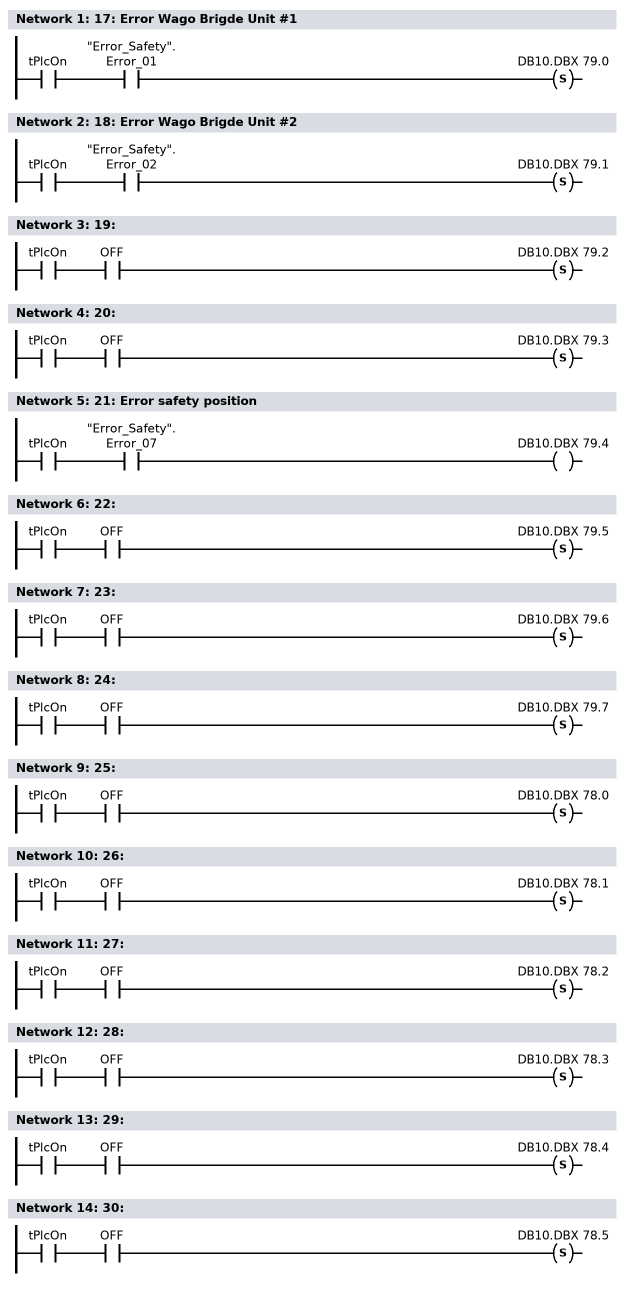
[picture p24: Errors_017-032_GEN2 networks 1-14]
NETWORK
TITLE = 17: Error Wago Brigde Unit #1
      A     "tPlcOn";
      A     "Error_Safety".Error_01;
      S     DB10.DBX 79.0;
NETWORK
TITLE = 18: Error Wago Brigde Unit #2
      A     "tPlcOn";
      A     "Error_Safety".Error_02;
      S     DB10.DBX 79.1;
NETWORK
TITLE = 19:
      A     "tPlcOn";
      A     "OFF";
      S     DB10.DBX 79.2;
NETWORK
TITLE = 20:
      A     "tPlcOn";
      A     "OFF";
      S     DB10.DBX 79.3;
NETWORK
TITLE = 21: Error safety position
      A     "tPlcOn";
      A     "Error_Safety".Error_07;
      =     DB10.DBX 79.4;
NETWORK
TITLE = 22:
      A     "tPlcOn";
      A     "OFF";
      S     DB10.DBX 79.5;
NETWORK
TITLE = 23:
      A     "tPlcOn";
      A     "OFF";
      S     DB10.DBX 79.6;
NETWORK
TITLE = 24:
      A     "tPlcOn";
      A     "OFF";
      S     DB10.DBX 79.7;
NETWORK
TITLE = 25:
      A     "tPlcOn";
      A     "OFF";
      S     DB10.DBX 78.0;
NETWORK
TITLE = 26:
      A     "tPlcOn";
      A     "OFF";
      S     DB10.DBX 78.1;
NETWORK
TITLE = 27:
      A     "tPlcOn";
      A     "OFF";
      S     DB10.DBX 78.2;
NETWORK
TITLE = 28:
      A     "tPlcOn";
      A     "OFF";
      S     DB10.DBX 78.3;
NETWORK
TITLE = 29:
      A     "tPlcOn";
      A     "OFF";
      S     DB10.DBX 78.4;
NETWORK
TITLE = 30:
      A     "tPlcOn";
      A     "OFF";
      S     DB10.DBX 78.5;
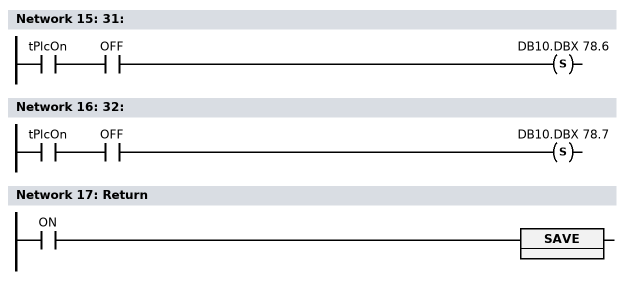
NETWORK
TITLE = 31:
      A     "tPlcOn";
      A     "OFF";
      S     DB10.DBX 78.6;
NETWORK
TITLE = 32:
      A     "tPlcOn";
      A     "OFF";
      S     DB10.DBX 78.7;
NETWORK
TITLE = Return
      A     "ON";
      SAVE;
END_FUNCTION

FUNCTION "Errors_033-048_NET" : VOID	// FC 44
TITLE = Errors NET
VERSION : 0.1
BEGIN
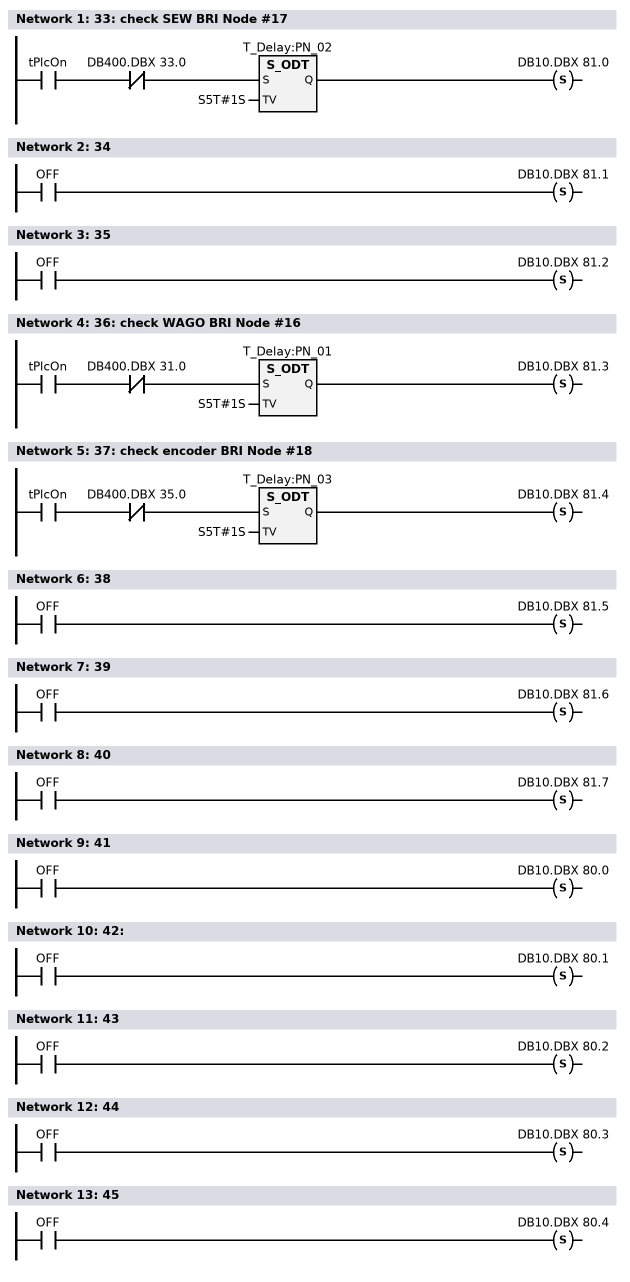
NETWORK
TITLE = 33: check SEW BRI Node #17
      A     "tPlcOn";
      AN    DB400.DBX 33.0;
      L     S5T#1S;
      SD    "T_Delay:PN_02";
      NOP   0;
      NOP   0;
      NOP   0;
      A     "T_Delay:PN_02";
      S     DB10.DBX 81.0;
NETWORK
TITLE = 34
      A     "OFF";
      S     DB10.DBX 81.1;
NETWORK
TITLE = 35
      A     "OFF";
      S     DB10.DBX 81.2;
NETWORK
TITLE = 36: check WAGO BRI Node #16
      A     "tPlcOn";
      AN    DB400.DBX 31.0;
      L     S5T#1S;
      SD    "T_Delay:PN_01";
      NOP   0;
      NOP   0;
      NOP   0;
      A     "T_Delay:PN_01";
      S     DB10.DBX 81.3;
NETWORK
TITLE = 37: check encoder BRI Node #18
      A     "tPlcOn";
      AN    DB400.DBX 35.0;
      L     S5T#1S;
      SD    "T_Delay:PN_03";
      NOP   0;
      NOP   0;
      NOP   0;
      A     "T_Delay:PN_03";
      S     DB10.DBX 81.4;
NETWORK
TITLE = 38
      A     "OFF";
      S     DB10.DBX 81.5;
NETWORK
TITLE = 39
      A     "OFF";
      S     DB10.DBX 81.6;
NETWORK
TITLE = 40
      A     "OFF";
      S     DB10.DBX 81.7;
NETWORK
TITLE = 41
      A     "OFF";
      S     DB10.DBX 80.0;
NETWORK
TITLE = 42:
      A     "OFF";
      S     DB10.DBX 80.1;
NETWORK
TITLE = 43
      A     "OFF";
      S     DB10.DBX 80.2;
NETWORK
TITLE = 44
      A     "OFF";
      S     DB10.DBX 80.3;
NETWORK
TITLE = 45
      A     "OFF";
      S     DB10.DBX 80.4;
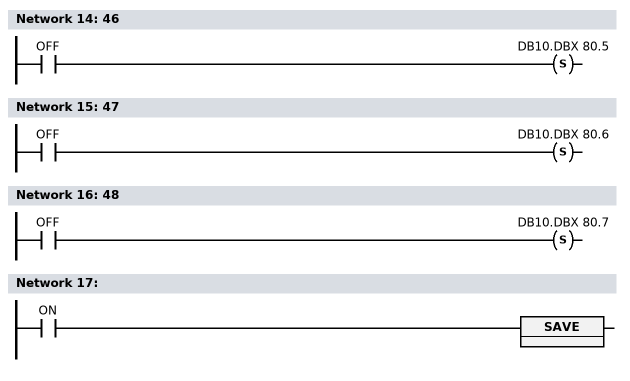
NETWORK
TITLE = 46
      A     "OFF";
      S     DB10.DBX 80.5;
NETWORK
TITLE = 47
      A     "OFF";
      S     DB10.DBX 80.6;
NETWORK
TITLE = 48
      A     "OFF";
      S     DB10.DBX 80.7;
NETWORK
TITLE =
      A     "ON";
      SAVE;
END_FUNCTION

FUNCTION "EOff_MachineOff" : VOID	// FC 48
TITLE = EOff Machine off
//TODO disable the remote in auto
VERSION : 0.1
VAR_TEMP
  INT_DivEoff : BOOL ;
  INT_Err_GEN1 : BOOL ;
  INT_Err_GEN2 : BOOL ;
  INT_Err_NET : BOOL ;
  INT_Err_BRI : BOOL ;
  INT_Err_TRO : BOOL ;
  INT_Err_LIF : BOOL ;
  INT_Err_TEL : BOOL ;
  INT_Warn : BOOL ;
  INT_OPM1 : BOOL ;
  INT_OPM2 : BOOL ;
  INT_ERR_06 : BOOL ;
  INT_ERR_07 : BOOL ;
  INT_ERR_08 : BOOL ;
  INT_ERR_09 : BOOL ;
  INT_ERR_10 : BOOL ;
  INT_ERR_11 : BOOL ;
  INT_MSG_01 : BOOL ;
  INT_MSG_02 : BOOL ;
  INT_MSG_03 : BOOL ;
  INT_MSG_04 : BOOL ;
  INT_MSG_05 : BOOL ;
END_VAR
BEGIN
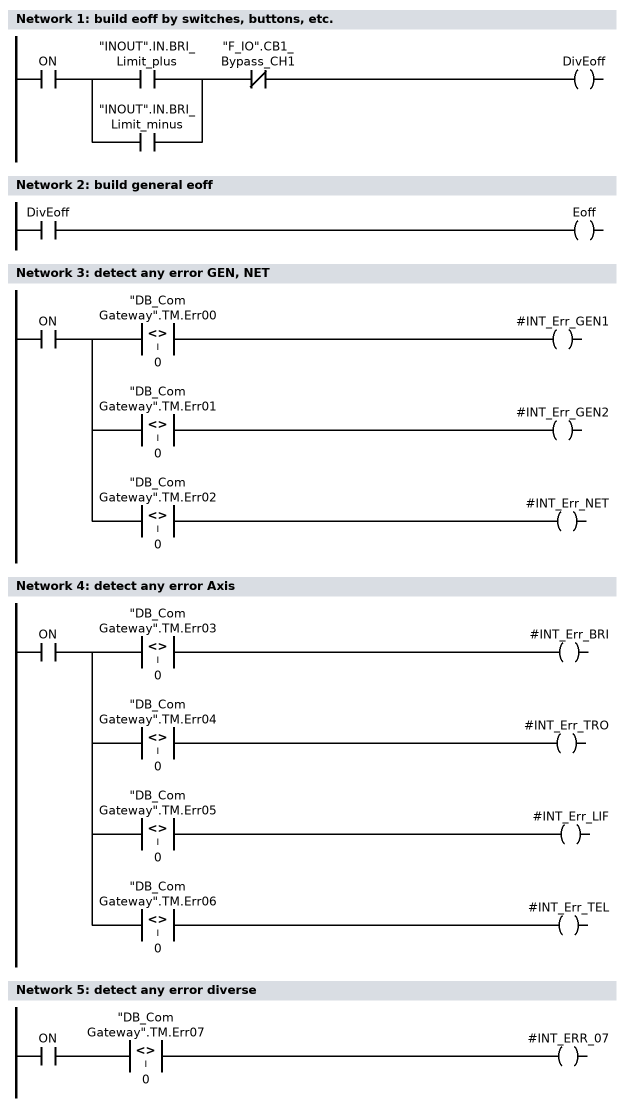
NETWORK
TITLE = build eoff by switches, buttons, etc.
      A     "ON";
      A(;
      O     "INOUT".IN.BRI_Limit_plus;
      O     "INOUT".IN.BRI_Limit_minus;
      );
      AN    "F_IO".CB1_Bypass_CH1;
      =     "DivEoff";
NETWORK
TITLE = build general eoff
      A     "DivEoff";
      =     "Eoff";
NETWORK
TITLE = detect any error GEN, NET
      A     "ON";
      =     L 3.0;
      A     L 3.0;
      A(;
      L     "DB_ComGateway".TM.Err00;
      L     0;
      <>I;
      );
      =     #INT_Err_GEN1;
      A     L 3.0;
      A(;
      L     "DB_ComGateway".TM.Err01;
      L     0;
      <>I;
      );
      =     #INT_Err_GEN2;
      A     L 3.0;
      A(;
      L     "DB_ComGateway".TM.Err02;
      L     0;
      <>I;
      );
      =     #INT_Err_NET;
NETWORK
TITLE = detect any error Axis
      A     "ON";
      =     L 3.0;
      A     L 3.0;
      A(;
      L     "DB_ComGateway".TM.Err03;
      L     0;
      <>I;
      );
      =     #INT_Err_BRI;
      A     L 3.0;
      A(;
      L     "DB_ComGateway".TM.Err04;
      L     0;
      <>I;
      );
      =     #INT_Err_TRO;
      A     L 3.0;
      A(;
      L     "DB_ComGateway".TM.Err05;
      L     0;
      <>I;
      );
      =     #INT_Err_LIF;
      A     L 3.0;
      A(;
      L     "DB_ComGateway".TM.Err06;
      L     0;
      <>I;
      );
      =     #INT_Err_TEL;
NETWORK
TITLE = detect any error diverse
      A     "ON";
      A(;
      L     "DB_ComGateway".TM.Err07;
      L     0;
      <>I;
      );
      =     #INT_ERR_07;
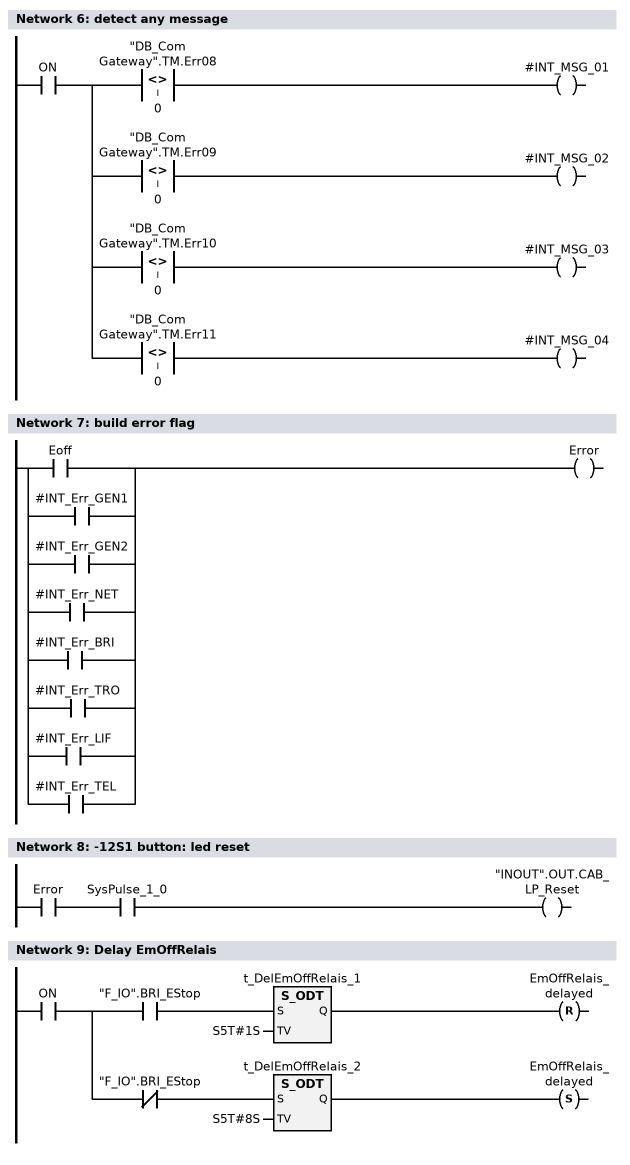
NETWORK
TITLE = detect any message
      A     "ON";
      =     L 3.0;
      A     L 3.0;
      A(;
      L     "DB_ComGateway".TM.Err08;
      L     0;
      <>I;
      );
      =     #INT_MSG_01;
      A     L 3.0;
      A(;
      L     "DB_ComGateway".TM.Err09;
      L     0;
      <>I;
      );
      =     #INT_MSG_02;
      A     L 3.0;
      A(;
      L     "DB_ComGateway".TM.Err10;
      L     0;
      <>I;
      );
      =     #INT_MSG_03;
      A     L 3.0;
      A(;
      L     "DB_ComGateway".TM.Err11;
      L     0;
      <>I;
      );
      =     #INT_MSG_04;
NETWORK
TITLE = build error flag
//xOff for error words
//
      O     "Eoff";
      O     #INT_Err_GEN1;
      O     #INT_Err_GEN2;
      O     #INT_Err_NET;
      O     #INT_Err_BRI;
      O     #INT_Err_TRO;
      O     #INT_Err_LIF;
      O     #INT_Err_TEL;
      =     "Error";
NETWORK
TITLE = -12S1 button: led reset
      A     "Error";
      A     "SysPulse_1_0";
      =     "INOUT".OUT.CAB_LP_Reset;
NETWORK
TITLE = Delay EmOffRelais
      A     "ON";
      =     L 3.0;
      A     L 3.0;
      A     "F_IO".BRI_EStop;
      L     S5T#1S;
      SD    "t_DelEmOffRelais_1";
      NOP   0;
      NOP   0;
      NOP   0;
      A     "t_DelEmOffRelais_1";
      R     "EmOffRelais_delayed";
      A     L 3.0;
      AN    "F_IO".BRI_EStop;
      L     S5T#8S;
      SD    "t_DelEmOffRelais_2";
      NOP   0;
      NOP   0;
      NOP   0;
      A     "t_DelEmOffRelais_2";
      S     "EmOffRelais_delayed";
END_FUNCTION

FUNCTION "OP_Mode" : VOID	// FC 49
TITLE = OP Mode
VERSION : 0.1
VAR_TEMP
  TEMP_DINT_00 : DINT ;
  TEMP_DINT_01 : DINT ;
  TEMP_BOOL_00 : BOOL ;
  TEMP_BOOL_01 : BOOL ;
  TEMP_BOOL_02 : BOOL ;
  TEMP_BOOL_03 : BOOL ;
  TEMP_BOOL_04 : BOOL ;
  TEMP_BOOL_05 : BOOL ;
  TEMP_BOOL_06 : BOOL ;
  value : INT ;
  lampPrio : INT ;
  Encoder : DINT ;
END_VAR
BEGIN
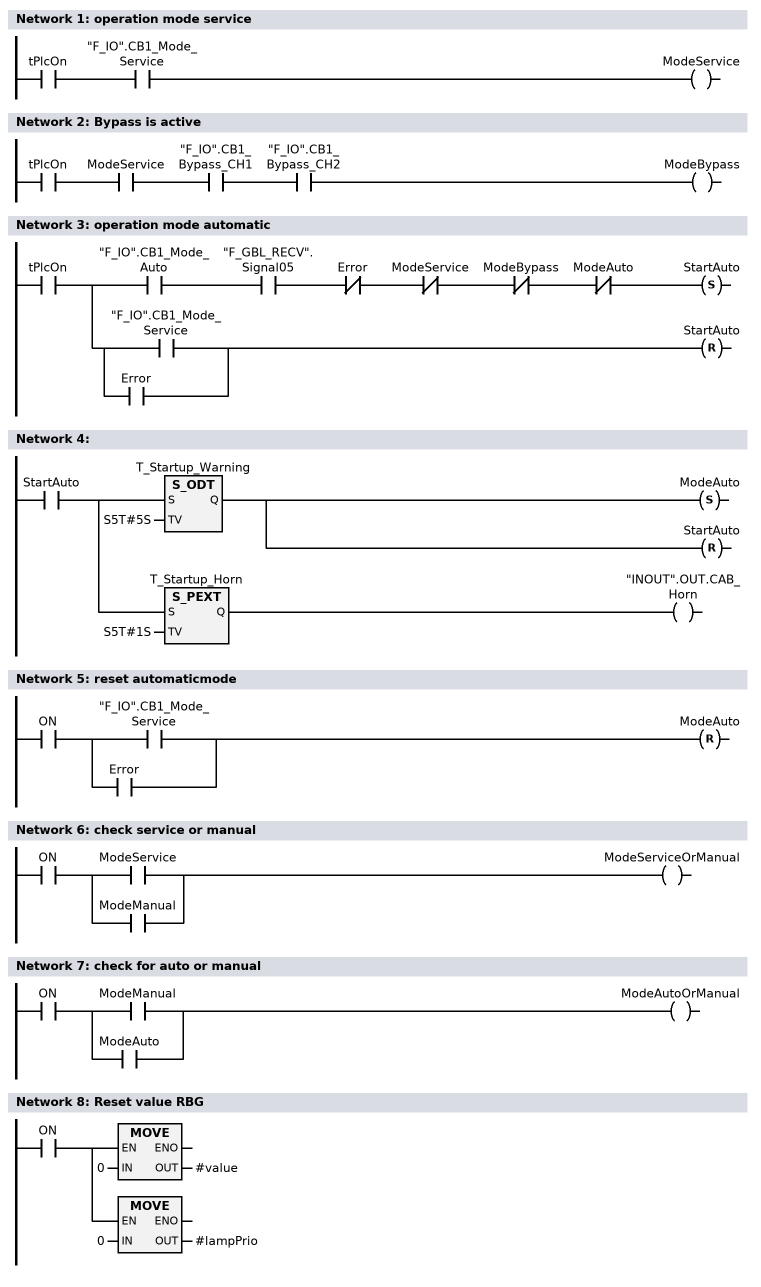
NETWORK
TITLE = operation mode service
      A     "tPlcOn";
      A     "F_IO".CB1_Mode_Service;
      =     "ModeService";
NETWORK
TITLE = Bypass is active
      A     "tPlcOn";
      A     "ModeService";
      A     "F_IO".CB1_Bypass_CH1;
      A     "F_IO".CB1_Bypass_CH2;
      =     "ModeBypass";
NETWORK
TITLE = operation mode automatic
      A     "tPlcOn";
      =     L 18.0;
      A     L 18.0;
      A     "F_IO".CB1_Mode_Auto;
      A     "F_GBL_RECV".Signal05;
      AN    "Error";
      AN    "ModeService";
      AN    "ModeBypass";
      AN    "ModeAuto";
      S     "StartAuto";
      A     L 18.0;
      A(;
      O     "F_IO".CB1_Mode_Service;
      O     "Error";
      );
      R     "StartAuto";
NETWORK
TITLE =
      A     "StartAuto";
      =     L 18.0;
      A     L 18.0;
      L     S5T#5S;
      SD    "T_Startup_Warning";
      NOP   0;
      NOP   0;
      NOP   0;
      A     "T_Startup_Warning";
      S     "ModeAuto";
      R     "StartAuto";
      A     L 18.0;
      L     S5T#1S;
      SE    "T_Startup_Horn";
      NOP   0;
      NOP   0;
      NOP   0;
      A     "T_Startup_Horn";
      =     "INOUT".OUT.CAB_Horn;
NETWORK
TITLE = reset automaticmode
      A     "ON";
      A(;
      O     "F_IO".CB1_Mode_Service;
      O     "Error";
      );
      R     "ModeAuto";
NETWORK
TITLE = check service or manual
      A     "ON";
      A(;
      O     "ModeService";
      O     "ModeManual";
      );
      =     "ModeServiceOrManual";
NETWORK
TITLE = check for auto or manual
      A     "ON";
      A(;
      O     "ModeManual";
      O     "ModeAuto";
      );
      =     "ModeAutoOrManual";
NETWORK
TITLE = Reset value RBG
      A     "ON";
      =     L 18.0;
      A     L 18.0;
      JNB   _001;
      L     0;
      T     #value;
_001: NOP   0;
      A     L 18.0;
      JNB   _002;
      L     0;
      T     #lampPrio;
_002: NOP   0;
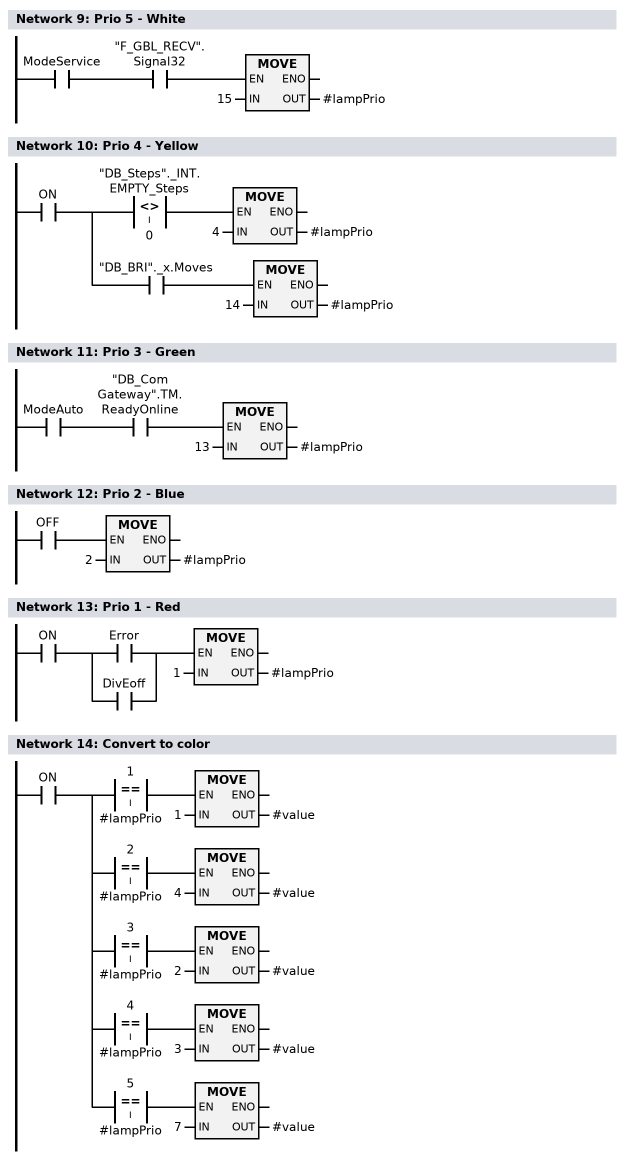
NETWORK
TITLE = Prio 5 - White
      A     "ModeService";
      A     "F_GBL_RECV".Signal32;
      JNB   _003;
      L     15;
      T     #lampPrio;
_003: NOP   0;
NETWORK
TITLE = Prio 4 - Yellow
      A     "ON";
      =     L 18.0;
      A     L 18.0;
      A(;
      L     "DB_Steps"._INT.EMPTY_Steps;
      L     0;
      <>I;
      );
      JNB   _004;
      L     4;
      T     #lampPrio;
_004: NOP   0;
      A     L 18.0;
      A     "DB_BRI"._x.Moves;
      JNB   _005;
      L     14;
      T     #lampPrio;
_005: NOP   0;
NETWORK
TITLE = Prio 3 - Green
      A     "ModeAuto";
      A     "DB_ComGateway".TM.ReadyOnline;
      JNB   _006;
      L     13;
      T     #lampPrio;
_006: NOP   0;
NETWORK
TITLE = Prio 2 - Blue
      A     "OFF";
      JNB   _007;
      L     2;
      T     #lampPrio;
_007: NOP   0;
NETWORK
TITLE = Prio 1 - Red
      A     "ON";
      A(;
      O     "Error";
      O     "DivEoff";
      );
      JNB   _008;
      L     1;
      T     #lampPrio;
_008: NOP   0;
NETWORK
TITLE = Convert to color
      A     "ON";
      =     L 18.0;
      A     L 18.0;
      A(;
      L     1;
      L     #lampPrio;
      ==I;
      );
      JNB   _009;
      L     1;
      T     #value;
_009: NOP   0;
      A     L 18.0;
      A(;
      L     2;
      L     #lampPrio;
      ==I;
      );
      JNB   _00a;
      L     4;
      T     #value;
_00a: NOP   0;
      A     L 18.0;
      A(;
      L     3;
      L     #lampPrio;
      ==I;
      );
      JNB   _00b;
      L     2;
      T     #value;
_00b: NOP   0;
      A     L 18.0;
      A(;
      L     4;
      L     #lampPrio;
      ==I;
      );
      JNB   _00c;
      L     3;
      T     #value;
_00c: NOP   0;
      A     L 18.0;
      A(;
      L     5;
      L     #lampPrio;
      ==I;
      );
      JNB   _00d;
      L     7;
      T     #value;
_00d: NOP   0;
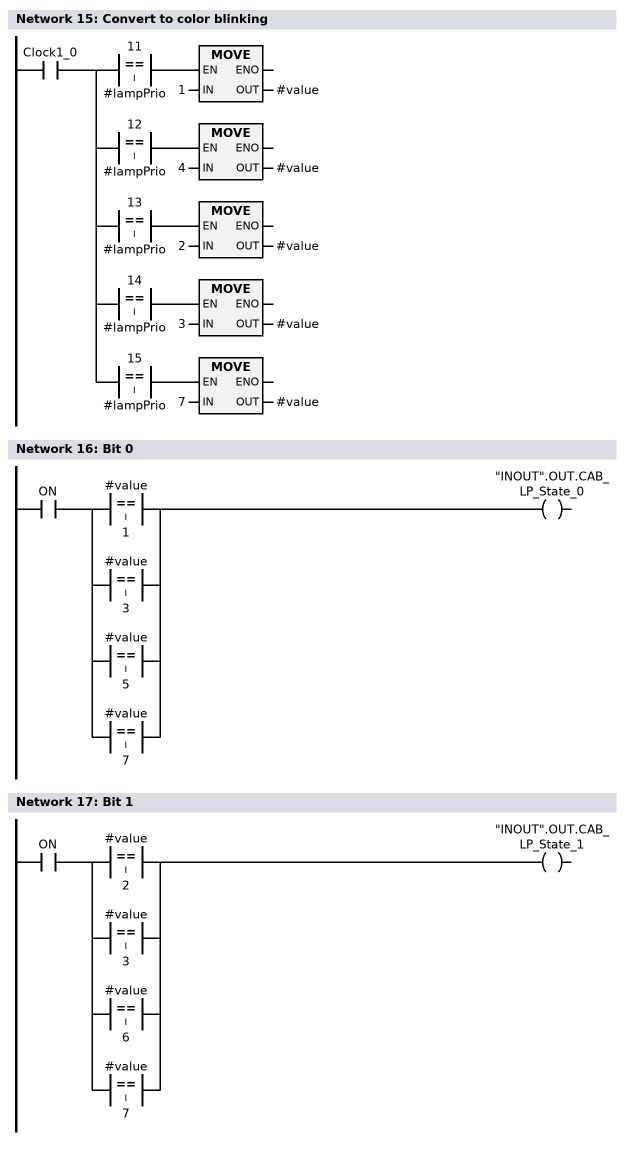
NETWORK
TITLE = Convert to color blinking
      A     "Clock1_0";
      =     L 18.0;
      A     L 18.0;
      A(;
      L     11;
      L     #lampPrio;
      ==I;
      );
      JNB   _00e;
      L     1;
      T     #value;
_00e: NOP   0;
      A     L 18.0;
      A(;
      L     12;
      L     #lampPrio;
      ==I;
      );
      JNB   _00f;
      L     4;
      T     #value;
_00f: NOP   0;
      A     L 18.0;
      A(;
      L     13;
      L     #lampPrio;
      ==I;
      );
      JNB   _010;
      L     2;
      T     #value;
_010: NOP   0;
      A     L 18.0;
      A(;
      L     14;
      L     #lampPrio;
      ==I;
      );
      JNB   _011;
      L     3;
      T     #value;
_011: NOP   0;
      A     L 18.0;
      A(;
      L     15;
      L     #lampPrio;
      ==I;
      );
      JNB   _012;
      L     7;
      T     #value;
_012: NOP   0;
NETWORK
TITLE = Bit 0
//BIT 0 1 2 Color
//-----------------
//0    0 0 0 Off
//1    1 0 0 red
//2    0 1 0 green
//3    1 1 0 yellow
//4    0 0 1 blue
//5    1 0 1 viloet 
//6    0 1 1 turque
//7    1 1 1 white
      A     "ON";
      A(;
      O(;
      L     #value;
      L     1;
      ==I;
      );
      O(;
      L     #value;
      L     3;
      ==I;
      );
      O(;
      L     #value;
      L     5;
      ==I;
      );
      O(;
      L     #value;
      L     7;
      ==I;
      );
      );
      =     "INOUT".OUT.CAB_LP_State_0;
NETWORK
TITLE = Bit 1
      A     "ON";
      A(;
      O(;
      L     #value;
      L     2;
      ==I;
      );
      O(;
      L     #value;
      L     3;
      ==I;
      );
      O(;
      L     #value;
      L     6;
      ==I;
      );
      O(;
      L     #value;
      L     7;
      ==I;
      );
      );
      =     "INOUT".OUT.CAB_LP_State_1;
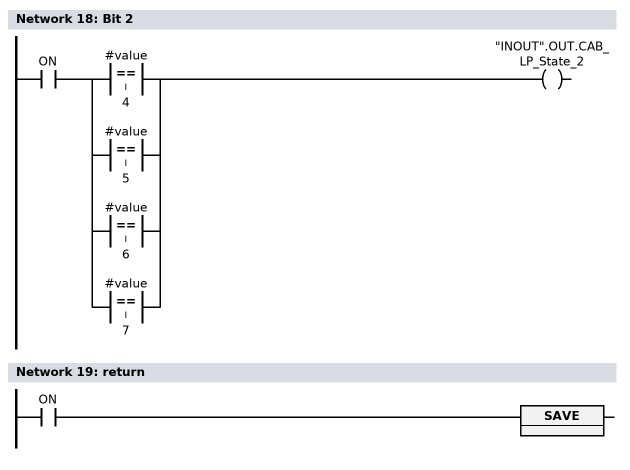
NETWORK
TITLE = Bit 2
      A     "ON";
      A(;
      O(;
      L     #value;
      L     4;
      ==I;
      );
      O(;
      L     #value;
      L     5;
      ==I;
      );
      O(;
      L     #value;
      L     6;
      ==I;
      );
      O(;
      L     #value;
      L     7;
      ==I;
      );
      );
      =     "INOUT".OUT.CAB_LP_State_2;
NETWORK
TITLE = return
      A     "ON";
      SAVE;
END_FUNCTION

FUNCTION "Send_Buffer" : VOID	// FC 52
TITLE = Handle Buffer
VERSION : 0.1
VAR_TEMP
  Count : INT ;
  POINT1 : DWORD ;
  POINT2 : DWORD ;
  POINT3 : DWORD ;
  POINT4 : DWORD ;
  Data : BOOL ;
  Space : BOOL ;
  Loop : INT ;
  Return : INT ;
END_VAR
BEGIN
NETWORK
TITLE = Init values
      L     0;
      T     #Count;
      L     L#52;
      SLD   3;
      T     #POINT1;
      L     L#26;
      SLD   3;
      T     #POINT2;
      OPN   "Moves";
l0:   NOP   0;	// Start of main loop
NETWORK
TITLE = Check for Data
      L     DBW [#POINT1];
      L     0;
      <>I;
      =     #Data;
NETWORK
TITLE = Check for Space
      L     DBW [#POINT2];
      L     0;
      ==I;
      =     #Space;
NETWORK
TITLE = Copy up
      A     #Data;
      A     #Space;
      JCN   m0;
      L     #POINT1;
      T     #POINT3;
      L     #POINT2;
      T     #POINT4;
      L     0;
      T     #Loop;
mm:   L     DBW [#POINT3];
      T     DBW [#POINT4];
      L     0;
      T     DBW [#POINT3];
      L     #POINT3;
      L     L#16;
      +D;
      T     #POINT3;
      L     #POINT4;
      L     L#16;
      +D;
      T     #POINT4;
      L     #Loop;
      L     1;
      +I;
      T     #Loop;
      L     13;
      <I;
      JC    mm;
m0:   NOP   0;
NETWORK
TITLE = Next loop ?
      L     #POINT1;
      SRD   3;
      L     L#26;
      +D;
      SLD   3;
      T     #POINT1;
      L     #POINT2;
      SRD   3;
      L     L#26;
      +D;
      SLD   3;
      T     #POINT2;
      L     #Count;
      L     1;
      +I;
      T     #Count;
      L     49;
      >=I;
      JCN   l0;
NETWORK
TITLE =
      SET;
      SAVE;
END_FUNCTION

FUNCTION "MSG_161-176" : VOID	// FC 55
TITLE = Messages 161 - 176
AUTHOR : Koenig
VERSION : 0.1
BEGIN
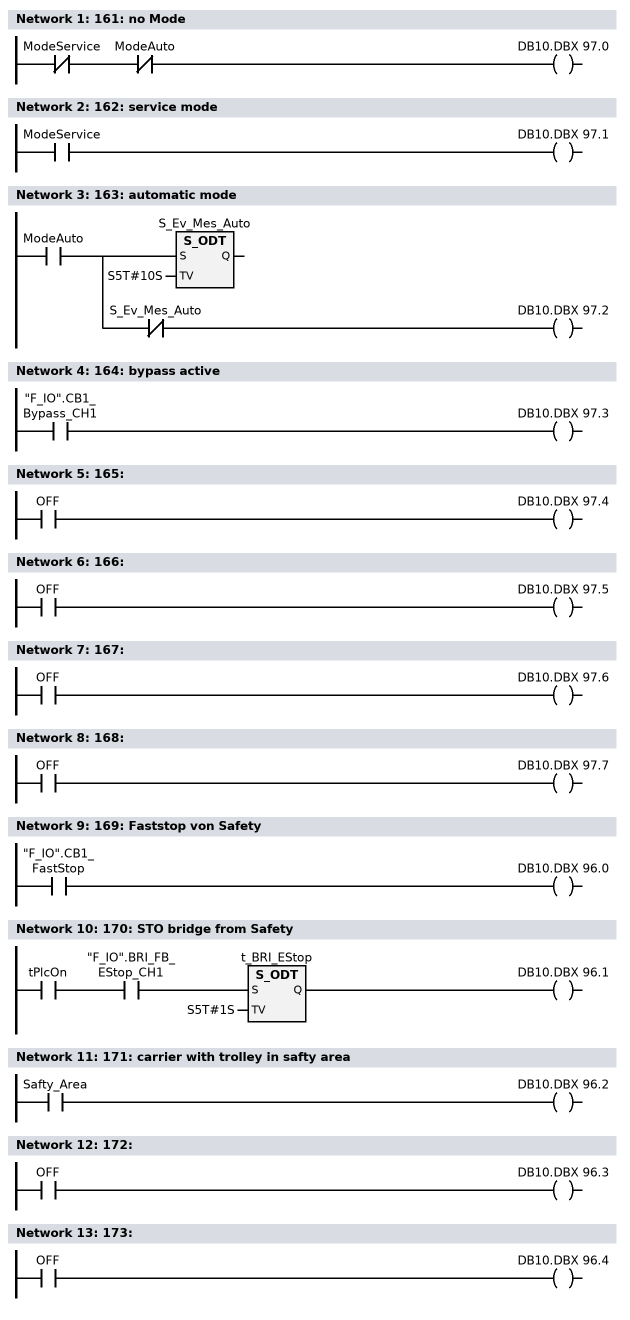
NETWORK
TITLE = 161: no Mode
      AN    "ModeService";
      AN    "ModeAuto";
      =     DB10.DBX 97.0;
NETWORK
TITLE = 162: service mode
      A     "ModeService";
      =     DB10.DBX 97.1;
NETWORK
TITLE = 163: automatic mode
      A     "ModeAuto";
      =     L 0.0;
      A     L 0.0;
      L     S5T#10S;
      SD    "S_Ev_Mes_Auto";
      NOP   0;
      NOP   0;
      NOP   0;
      NOP   0;
      A     L 0.0;
      AN    "S_Ev_Mes_Auto";
      =     DB10.DBX 97.2;
NETWORK
TITLE = 164: bypass active
      A     "F_IO".CB1_Bypass_CH1;
      =     DB10.DBX 97.3;
NETWORK
TITLE = 165:
      A     "OFF";
      =     DB10.DBX 97.4;
NETWORK
TITLE = 166:
      A     "OFF";
      =     DB10.DBX 97.5;
NETWORK
TITLE = 167:
      A     "OFF";
      =     DB10.DBX 97.6;
NETWORK
TITLE = 168:
      A     "OFF";
      =     DB10.DBX 97.7;
NETWORK
TITLE = 169: Faststop von Safety
      A     "F_IO".CB1_FastStop;
      =     DB10.DBX 96.0;
NETWORK
TITLE = 170: STO bridge from Safety
      A     "tPlcOn";
      A     "F_IO".BRI_FB_EStop_CH1;
      L     S5T#1S;
      SD    "t_BRI_EStop";
      NOP   0;
      NOP   0;
      NOP   0;
      A     "t_BRI_EStop";
      =     DB10.DBX 96.1;
NETWORK
TITLE = 171: carrier with trolley in safty area
      A     "Safty_Area";
      =     DB10.DBX 96.2;
NETWORK
TITLE = 172:
      A     "OFF";
      =     DB10.DBX 96.3;
NETWORK
TITLE = 173:
      A     "OFF";
      =     DB10.DBX 96.4;
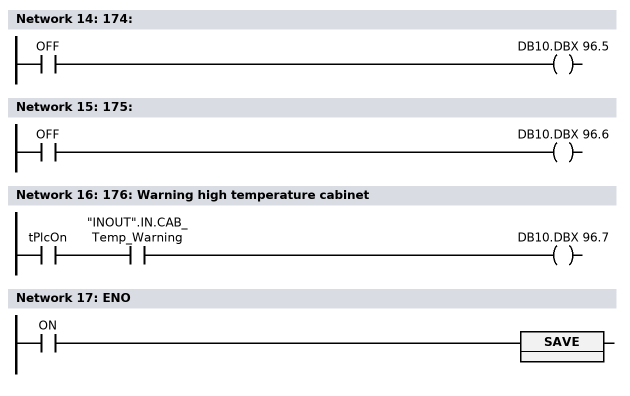
NETWORK
TITLE = 174:
      A     "OFF";
      =     DB10.DBX 96.5;
NETWORK
TITLE = 175:
      A     "OFF";
      =     DB10.DBX 96.6;
NETWORK
TITLE = 176: Warning high temperature cabinet
      A     "tPlcOn";
      A     "INOUT".IN.CAB_Temp_Warning;
      =     DB10.DBX 96.7;
NETWORK
TITLE = ENO
      A     "ON";
      SAVE;
END_FUNCTION

FUNCTION "MSG_177_192" : VOID	// FC 56
TITLE = Messages 177 - 192
AUTHOR : Koenig
VERSION : 0.1
BEGIN
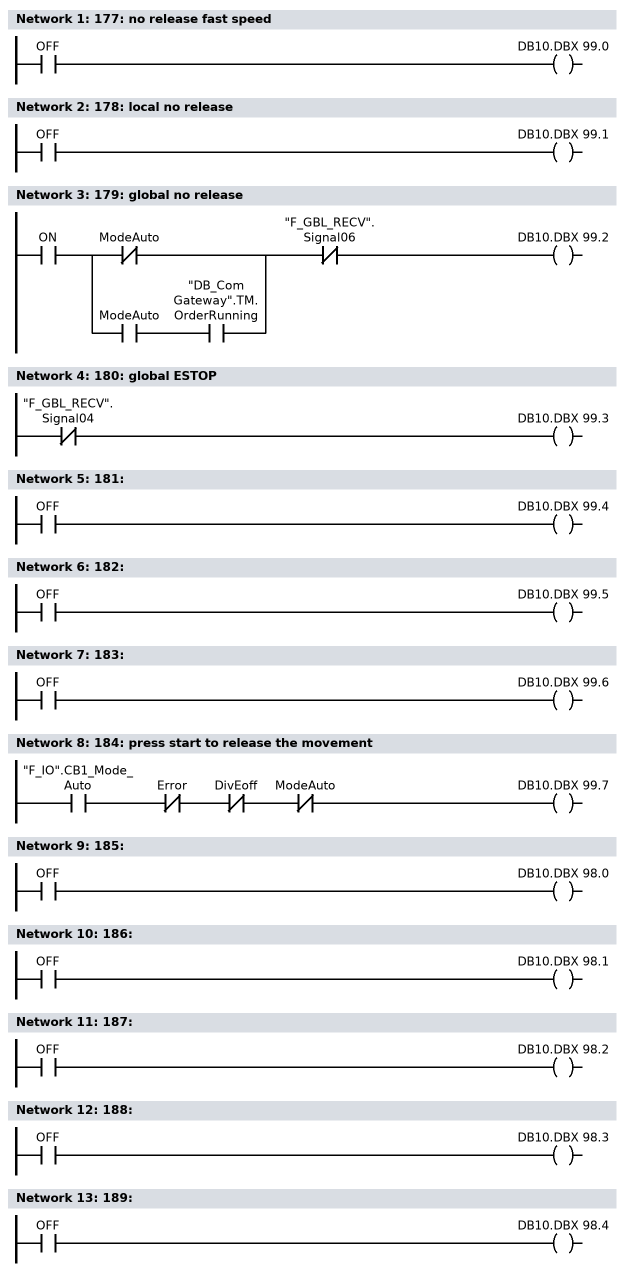
NETWORK
TITLE = 177: no release fast speed
      A     "OFF";
      =     DB10.DBX 99.0;
NETWORK
TITLE = 178: local no release
      A     "OFF";
      =     DB10.DBX 99.1;
NETWORK
TITLE = 179: global no release
      A     "ON";
      A(;
      ON    "ModeAuto";
      O;
      A     "ModeAuto";
      A     "DB_ComGateway".TM.OrderRunning;
      );
      AN    "F_GBL_RECV".Signal06;
      =     DB10.DBX 99.2;
NETWORK
TITLE = 180: global ESTOP
      AN    "F_GBL_RECV".Signal04;
      =     DB10.DBX 99.3;
NETWORK
TITLE = 181:
      A     "OFF";
      =     DB10.DBX 99.4;
NETWORK
TITLE = 182:
      A     "OFF";
      =     DB10.DBX 99.5;
NETWORK
TITLE = 183:
      A     "OFF";
      =     DB10.DBX 99.6;
NETWORK
TITLE = 184: press start to release the movement
      A     "F_IO".CB1_Mode_Auto;
      AN    "Error";
      AN    "DivEoff";
      AN    "ModeAuto";
      =     DB10.DBX 99.7;
NETWORK
TITLE = 185:
      A     "OFF";
      =     DB10.DBX 98.0;
NETWORK
TITLE = 186:
      A     "OFF";
      =     DB10.DBX 98.1;
NETWORK
TITLE = 187:
      A     "OFF";
      =     DB10.DBX 98.2;
NETWORK
TITLE = 188:
      A     "OFF";
      =     DB10.DBX 98.3;
NETWORK
TITLE = 189:
      A     "OFF";
      =     DB10.DBX 98.4;
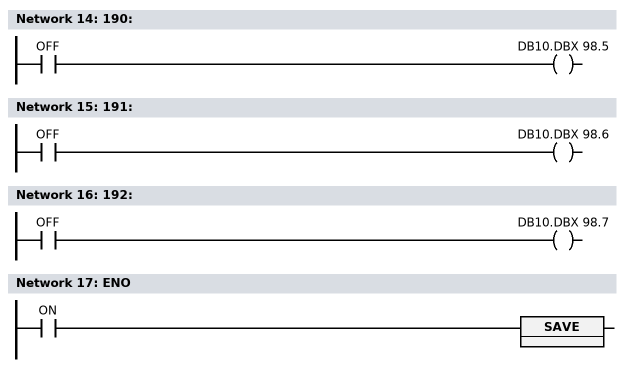
NETWORK
TITLE = 190:
      A     "OFF";
      =     DB10.DBX 98.5;
NETWORK
TITLE = 191:
      A     "OFF";
      =     DB10.DBX 98.6;
NETWORK
TITLE = 192:
      A     "OFF";
      =     DB10.DBX 98.7;
NETWORK
TITLE = ENO
      A     "ON";
      SAVE;
END_FUNCTION

FUNCTION "CheckWindowDi" : VOID	// FC 100
TITLE = Check Window
VERSION : 1.0
VAR_INPUT
  IN_diValue : DINT ;
  IN_diTestFor : DINT ;
  IN_diTolMinus : DINT ;
  IN_diTolPlus : DINT ;
END_VAR
VAR_OUTPUT
  OUT_xInWindow : BOOL ;
  OUT_udiAbsDiff : DINT ;
END_VAR
VAR_TEMP
  INT_diWinMinus : DINT ;
  INT_diWinPlus : DINT ;
  INT_xInWindow : BOOL ;
END_VAR
BEGIN
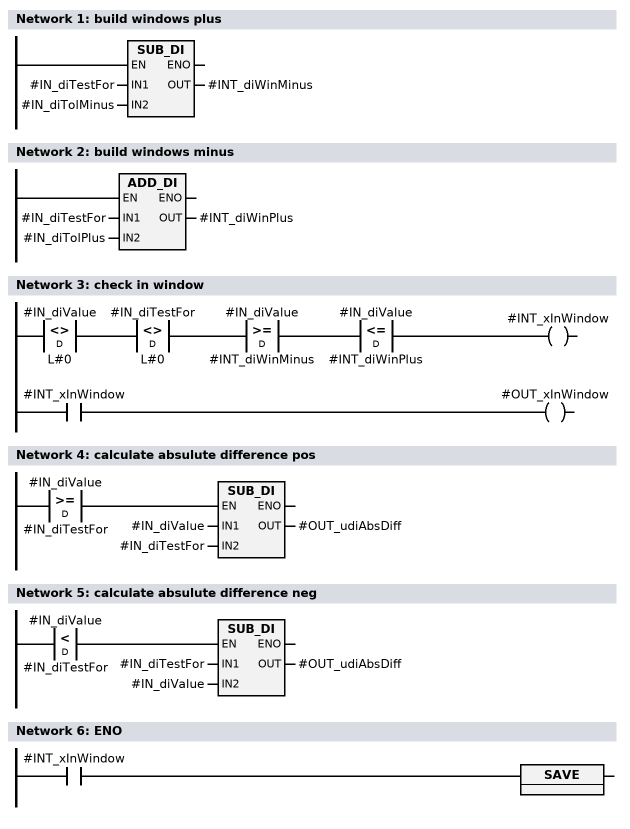
NETWORK
TITLE = build windows plus
      L     #IN_diTestFor;
      L     #IN_diTolMinus;
      -D;
      T     #INT_diWinMinus;
      NOP   0;
NETWORK
TITLE = build windows minus
      L     #IN_diTestFor;
      L     #IN_diTolPlus;
      +D;
      T     #INT_diWinPlus;
      NOP   0;
NETWORK
TITLE = check in window
      A(;
      L     #IN_diValue;
      L     L#0;
      <>D;
      );
      A(;
      L     #IN_diTestFor;
      L     L#0;
      <>D;
      );
      A(;
      L     #IN_diValue;
      L     #INT_diWinMinus;
      >=D;
      );
      A(;
      L     #IN_diValue;
      L     #INT_diWinPlus;
      <=D;
      );
      =     #INT_xInWindow;
      A     #INT_xInWindow;
      =     #OUT_xInWindow;
NETWORK
TITLE = calculate absulute difference pos
      A(;
      L     #IN_diValue;
      L     #IN_diTestFor;
      >=D;
      );
      JNB   _001;
      L     #IN_diValue;
      L     #IN_diTestFor;
      -D;
      T     #OUT_udiAbsDiff;
_001: NOP   0;
NETWORK
TITLE = calculate absulute difference neg
      A(;
      L     #IN_diValue;
      L     #IN_diTestFor;
      <D;
      );
      JNB   _002;
      L     #IN_diTestFor;
      L     #IN_diValue;
      -D;
      T     #OUT_udiAbsDiff;
_002: NOP   0;
NETWORK
TITLE = ENO
      A     #INT_xInWindow;
      SAVE;
END_FUNCTION

FUNCTION "Communication" : VOID	// FC 103
VERSION : 0.1
VAR_TEMP
  tmp_result : INT ;
  rel_online : BOOL ;
END_VAR
BEGIN
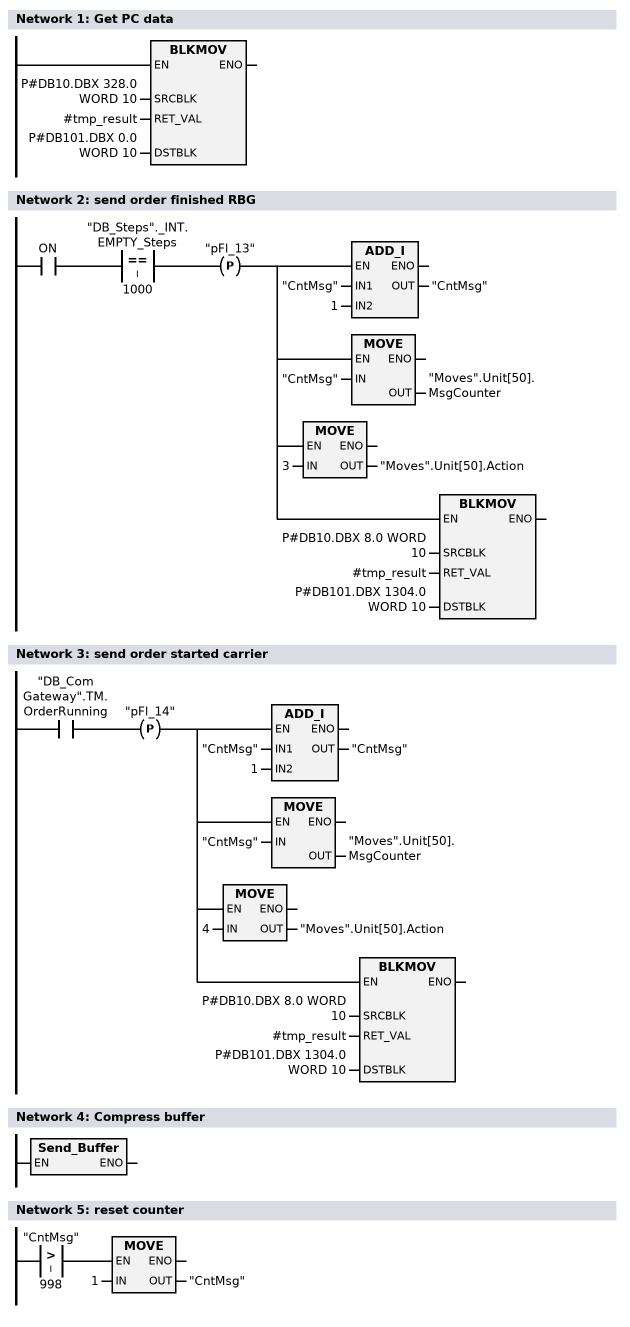
NETWORK
TITLE = Get PC data
      CALL  "BLKMOV" (
           SRCBLK                   := P#DB10.DBX 328.0 WORD 10,
           RET_VAL                  := #tmp_result,
           DSTBLK                   := P#DB101.DBX 0.0 WORD 10);
      NOP   0;
NETWORK
TITLE = send order finished RBG
      A     "ON";
      A(;
      L     "DB_Steps"._INT.EMPTY_Steps;
      L     1000;
      ==I;
      );
      FP    "pFl_13";
      =     L 3.0;
      A     L 3.0;
      JNB   _001;
      L     "CntMsg";
      L     1;
      +I;
      T     "CntMsg";
_001: NOP   0;
      A     L 3.0;
      JNB   _002;
      L     "CntMsg";
      T     "Moves".Unit[50].MsgCounter;
_002: NOP   0;
      A     L 3.0;
      JNB   _003;
      L     3;
      T     "Moves".Unit[50].Action;
_003: NOP   0;
      A     L 3.0;
      JNB   _004;
      CALL  "BLKMOV" (
           SRCBLK                   := P#DB10.DBX 8.0 WORD 10,
           RET_VAL                  := #tmp_result,
           DSTBLK                   := P#DB101.DBX 1304.0 WORD 10);
_004: NOP   0;
NETWORK
TITLE = send order started carrier
      A     "DB_ComGateway".TM.OrderRunning;
      FP    "pFl_14";
      =     L 3.0;
      A     L 3.0;
      JNB   _005;
      L     "CntMsg";
      L     1;
      +I;
      T     "CntMsg";
_005: NOP   0;
      A     L 3.0;
      JNB   _006;
      L     "CntMsg";
      T     "Moves".Unit[50].MsgCounter;
_006: NOP   0;
      A     L 3.0;
      JNB   _007;
      L     4;
      T     "Moves".Unit[50].Action;
_007: NOP   0;
      A     L 3.0;
      JNB   _008;
      CALL  "BLKMOV" (
           SRCBLK                   := P#DB10.DBX 8.0 WORD 10,
           RET_VAL                  := #tmp_result,
           DSTBLK                   := P#DB101.DBX 1304.0 WORD 10);
_008: NOP   0;
NETWORK
TITLE = Compress buffer
      CALL  "Send_Buffer";
      NOP   0;
NETWORK
TITLE = reset counter
      A(;
      L     "CntMsg";
      L     998;
      >I;
      );
      JNB   _009;
      L     1;
      T     "CntMsg";
_009: NOP   0;
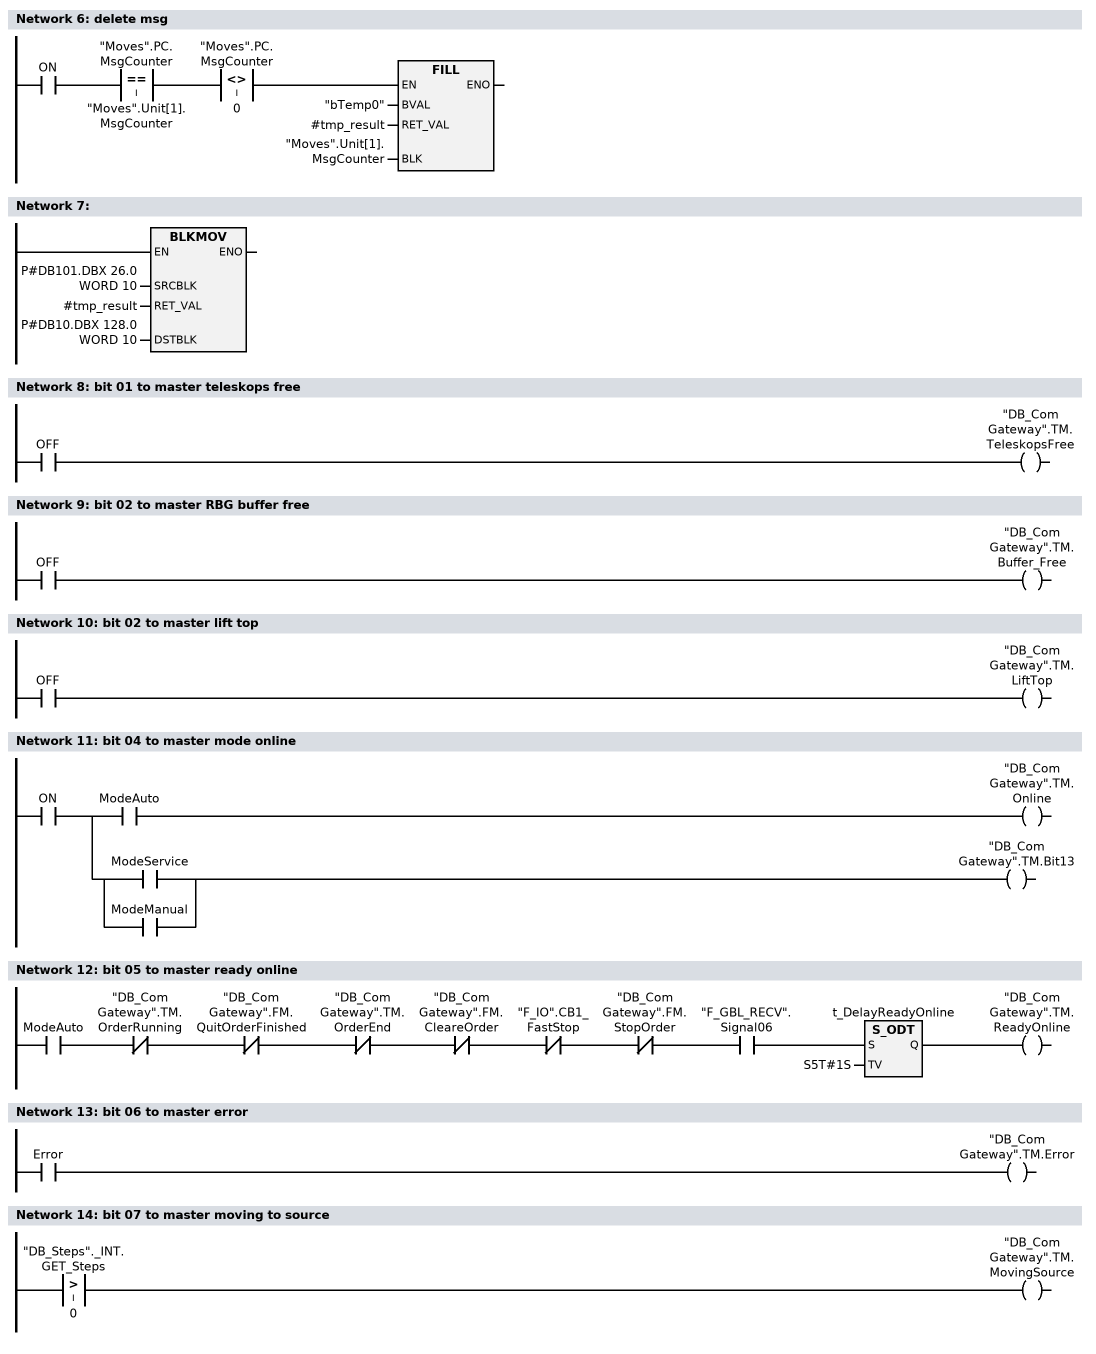
NETWORK
TITLE = delete msg
      A     "ON";
      A(;
      L     "Moves".PC.MsgCounter;
      L     "Moves".Unit[1].MsgCounter;
      ==I;
      );
      A(;
      L     "Moves".PC.MsgCounter;
      L     0;
      <>I;
      );
      JNB   _00a;
      CALL  "FILL" (
           BVAL                     := "bTemp0",
           RET_VAL                  := #tmp_result,
           BLK                      := "Moves".Unit[1].MsgCounter);
_00a: NOP   0;
NETWORK
TITLE =
      CALL  "BLKMOV" (
           SRCBLK                   := P#DB101.DBX 26.0 WORD 10,
           RET_VAL                  := #tmp_result,
           DSTBLK                   := P#DB10.DBX 128.0 WORD 10);
      NOP   0;
NETWORK
TITLE = bit 01 to master teleskops free
      A     "OFF";
      =     "DB_ComGateway".TM.TeleskopsFree;
NETWORK
TITLE = bit 02 to master RBG buffer free
      A     "OFF";
      =     "DB_ComGateway".TM.Buffer_Free;
NETWORK
TITLE = bit 02 to master lift top
      A     "OFF";
      =     "DB_ComGateway".TM.LiftTop;
NETWORK
TITLE = bit 04 to master mode online
      A     "ON";
      =     L 3.0;
      A     L 3.0;
      A     "ModeAuto";
      =     "DB_ComGateway".TM.Online;
      A     L 3.0;
      A(;
      O     "ModeService";
      O     "ModeManual";
      );
      =     "DB_ComGateway".TM.Bit13;
NETWORK
TITLE = bit 05 to master ready online
      A     "ModeAuto";
      AN    "DB_ComGateway".TM.OrderRunning;
      AN    "DB_ComGateway".FM.QuitOrderFinished;
      AN    "DB_ComGateway".TM.OrderEnd;
      AN    "DB_ComGateway".FM.CleareOrder;
      AN    "F_IO".CB1_FastStop;
      AN    "DB_ComGateway".FM.StopOrder;
      A     "F_GBL_RECV".Signal06;
      L     S5T#1S;
      SD    "t_DelayReadyOnline";
      NOP   0;
      NOP   0;
      NOP   0;
      A     "t_DelayReadyOnline";
      =     "DB_ComGateway".TM.ReadyOnline;
NETWORK
TITLE = bit 06 to master error
      A     "Error";
      =     "DB_ComGateway".TM.Error;
NETWORK
TITLE = bit 07 to master moving to source
      L     "DB_Steps"._INT.GET_Steps;
      L     0;
      >I;
      =     "DB_ComGateway".TM.MovingSource;
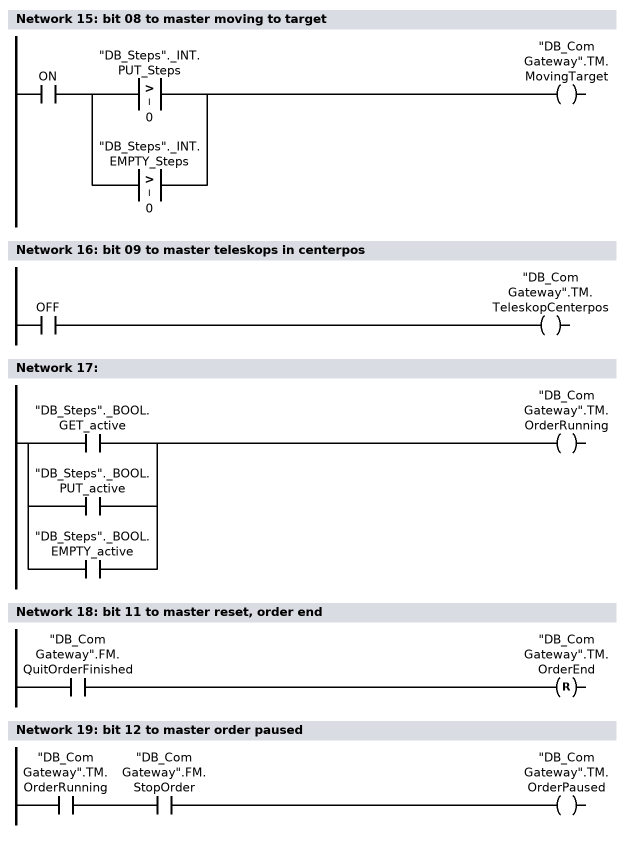
NETWORK
TITLE = bit 08 to master moving to target
      A     "ON";
      A(;
      O(;
      L     "DB_Steps"._INT.PUT_Steps;
      L     0;
      >I;
      );
      O(;
      L     "DB_Steps"._INT.EMPTY_Steps;
      L     0;
      >I;
      );
      );
      =     "DB_ComGateway".TM.MovingTarget;
NETWORK
TITLE = bit 09 to master teleskops in centerpos
      A     "OFF";
      =     "DB_ComGateway".TM.TeleskopCenterpos;
NETWORK
TITLE =
      O     "DB_Steps"._BOOL.GET_active;
      O     "DB_Steps"._BOOL.PUT_active;
      O     "DB_Steps"._BOOL.EMPTY_active;
      =     "DB_ComGateway".TM.OrderRunning;
NETWORK
TITLE = bit 11 to master reset, order end
      A     "DB_ComGateway".FM.QuitOrderFinished;
      R     "DB_ComGateway".TM.OrderEnd;
NETWORK
TITLE = bit 12 to master order paused
      A     "DB_ComGateway".TM.OrderRunning;
      A     "DB_ComGateway".FM.StopOrder;
      =     "DB_ComGateway".TM.OrderPaused;
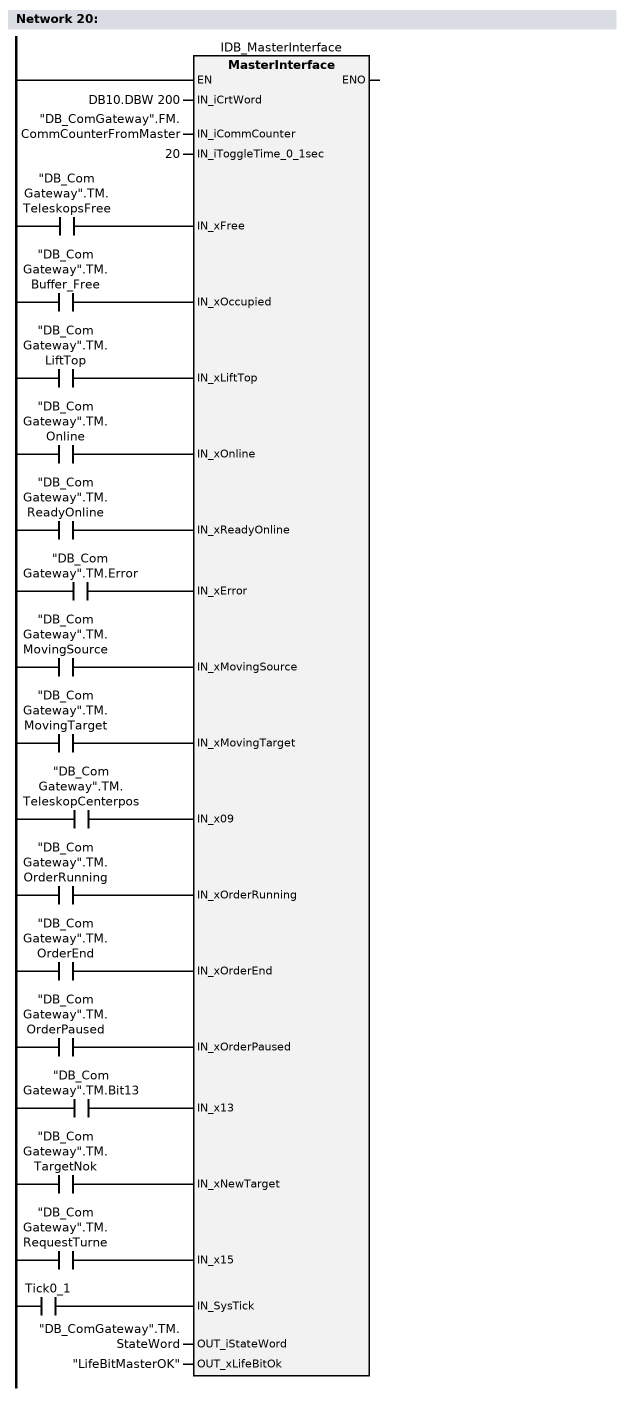
NETWORK
TITLE =
//we do not need the outputs....
//
      A     "DB_ComGateway".TM.TeleskopsFree;
      =     L 3.0;
      BLD   103;
      A     "DB_ComGateway".TM.Buffer_Free;
      =     L 3.1;
      BLD   103;
      A     "DB_ComGateway".TM.LiftTop;
      =     L 3.2;
      BLD   103;
      A     "DB_ComGateway".TM.Online;
      =     L 3.3;
      BLD   103;
      A     "DB_ComGateway".TM.ReadyOnline;
      =     L 3.4;
      BLD   103;
      A     "DB_ComGateway".TM.Error;
      =     L 3.5;
      BLD   103;
      A     "DB_ComGateway".TM.MovingSource;
      =     L 3.6;
      BLD   103;
      A     "DB_ComGateway".TM.MovingTarget;
      =     L 3.7;
      BLD   103;
      A     "DB_ComGateway".TM.TeleskopCenterpos;
      =     L 4.0;
      BLD   103;
      A     "DB_ComGateway".TM.OrderRunning;
      =     L 4.1;
      BLD   103;
      A     "DB_ComGateway".TM.OrderEnd;
      =     L 4.2;
      BLD   103;
      A     "DB_ComGateway".TM.OrderPaused;
      =     L 4.3;
      BLD   103;
      A     "DB_ComGateway".TM.Bit13;
      =     L 4.4;
      BLD   103;
      A     "DB_ComGateway".TM.TargetNok;
      =     L 4.5;
      BLD   103;
      A     "DB_ComGateway".TM.RequestTurne;
      =     L 4.6;
      BLD   103;
      A     "Tick0_1";
      =     L 4.7;
      BLD   103;
      CALL  "MasterInterface" , "IDB_MasterInterface" (
           IN_iCrtWord              := DB10.DBW 200,
           IN_iCommCounter          := "DB_ComGateway".FM.CommCounterFromMaster,
           IN_iToggleTime_0_1sec    := 20,
           IN_xFree                 := L 3.0,
           IN_xOccupied             := L 3.1,
           IN_xLiftTop              := L 3.2,
           IN_xOnline               := L 3.3,
           IN_xReadyOnline          := L 3.4,
           IN_xError                := L 3.5,
           IN_xMovingSource         := L 3.6,
           IN_xMovingTarget         := L 3.7,
           IN_x09                   := L 4.0,
           IN_xOrderRunning         := L 4.1,
           IN_xOrderEnd             := L 4.2,
           IN_xOrderPaused          := L 4.3,
           IN_x13                   := L 4.4,
           IN_xNewTarget            := L 4.5,
           IN_x15                   := L 4.6,
           IN_SysTick               := L 4.7,
           OUT_iStateWord           := "DB_ComGateway".TM.StateWord,
           OUT_xLifeBitOk           := "LifeBitMasterOK");
      NOP   0;
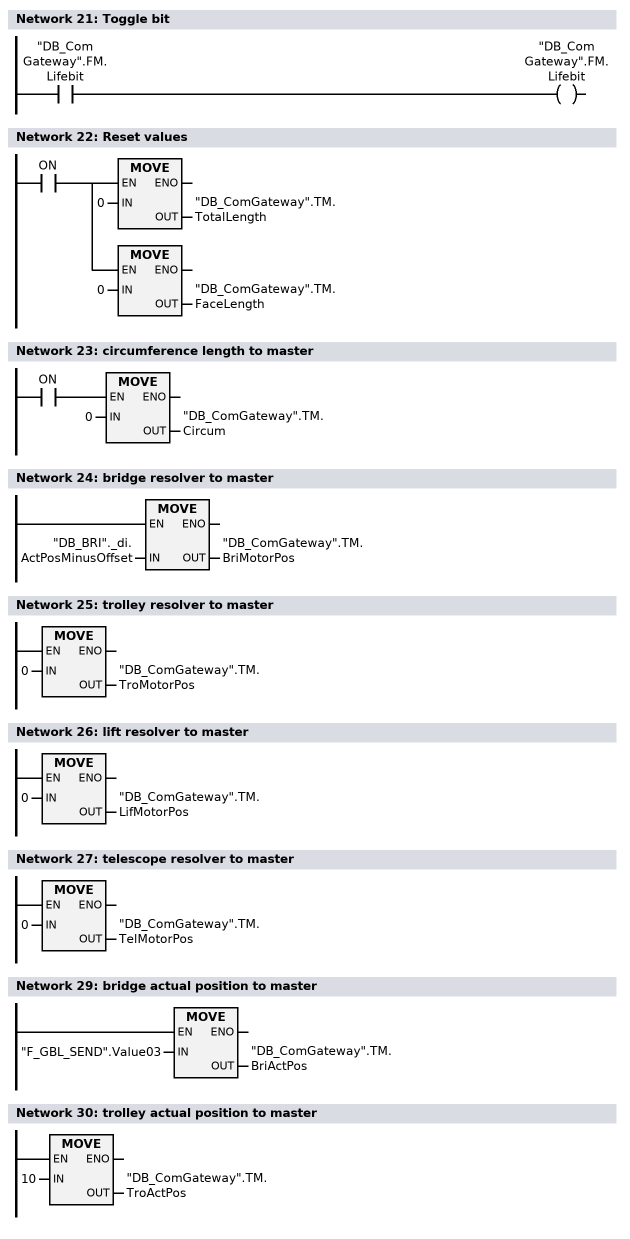
NETWORK
TITLE = Toggle bit
      A     "DB_ComGateway".FM.Lifebit;
      =     "DB_ComGateway".FM.Lifebit;
NETWORK
TITLE = Reset values
      A     "ON";
      =     L 3.0;
      A     L 3.0;
      JNB   _00b;
      L     0;
      T     "DB_ComGateway".TM.TotalLength;
_00b: NOP   0;
      A     L 3.0;
      JNB   _00c;
      L     0;
      T     "DB_ComGateway".TM.FaceLength;
_00c: NOP   0;
NETWORK
TITLE = circumference length to master
      A     "ON";
      JNB   _00d;
      L     0;
      T     "DB_ComGateway".TM.Circum;
_00d: NOP   0;
NETWORK
TITLE = bridge resolver to master
      L     "DB_BRI"._di.ActPosMinusOffset;
      T     "DB_ComGateway".TM.BriMotorPos;
      NOP   0;
NETWORK
TITLE = trolley resolver to master
      L     0;
      T     "DB_ComGateway".TM.TroMotorPos;
      NOP   0;
NETWORK
TITLE = lift resolver to master
      L     0;
      T     "DB_ComGateway".TM.LifMotorPos;
      NOP   0;
NETWORK
TITLE = telescope resolver to master
      L     0;
      T     "DB_ComGateway".TM.TelMotorPos;
      NOP   0;
NETWORK
TITLE = measured value to master
NETWORK
TITLE = bridge actual position to master
      L     "F_GBL_SEND".Value03;
      T     "DB_ComGateway".TM.BriActPos;
      NOP   0;
NETWORK
TITLE = trolley actual position to master
      L     10;
      T     "DB_ComGateway".TM.TroActPos;
      NOP   0;
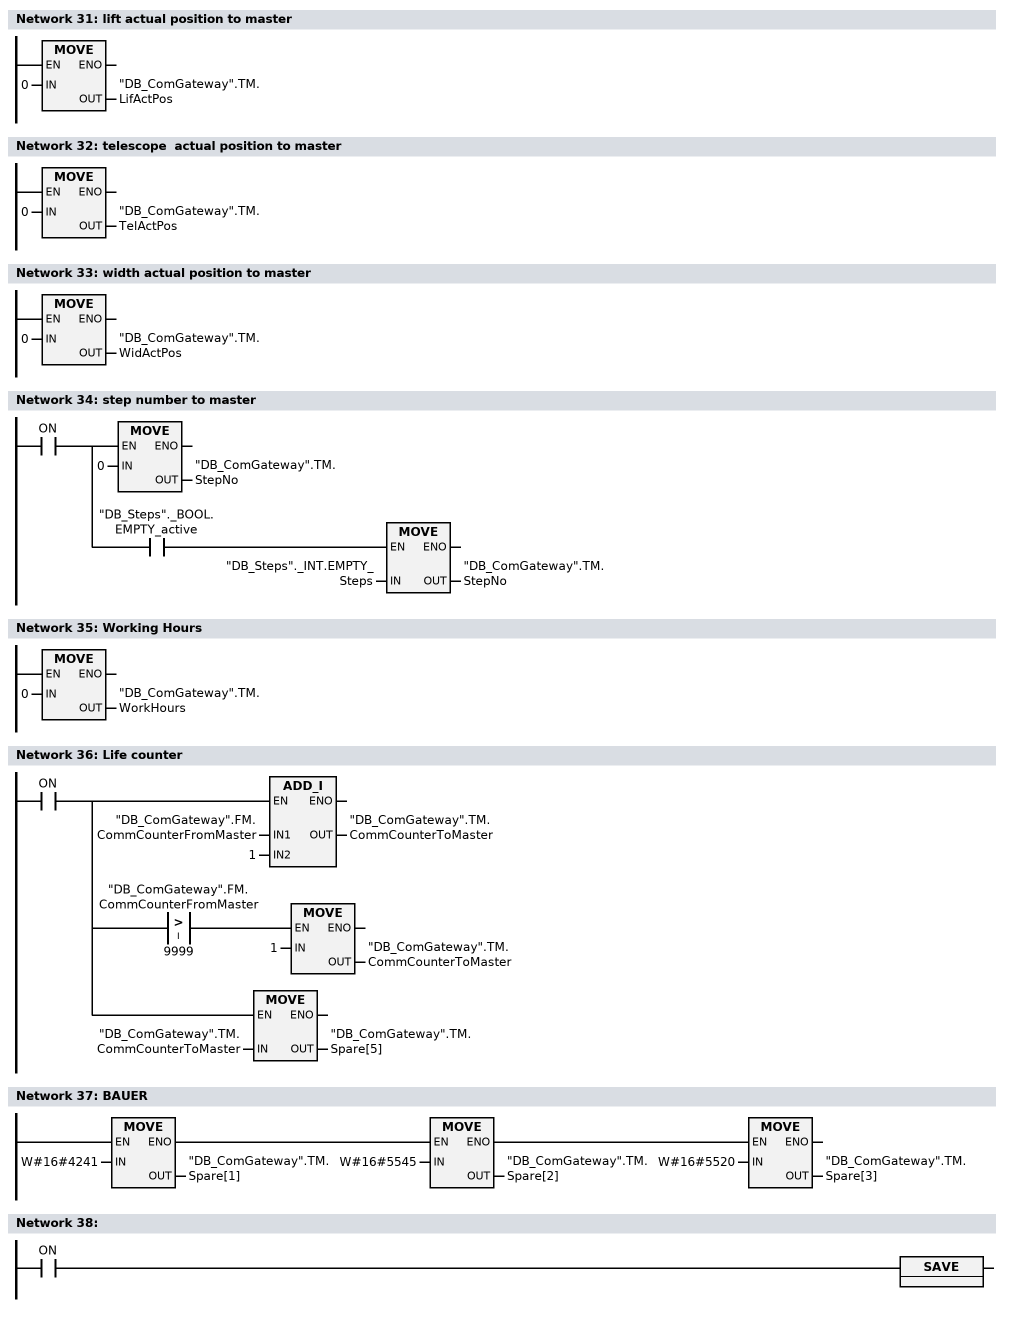
NETWORK
TITLE = lift actual position to master
      L     0;
      T     "DB_ComGateway".TM.LifActPos;
      NOP   0;
NETWORK
TITLE = telescope  actual position to master
      L     0;
      T     "DB_ComGateway".TM.TelActPos;
      NOP   0;
NETWORK
TITLE = width actual position to master
      L     0;
      T     "DB_ComGateway".TM.WidActPos;
      NOP   0;
NETWORK
TITLE = step number to master
      A     "ON";
      =     L 3.0;
      A     L 3.0;
      JNB   _00e;
      L     0;
      T     "DB_ComGateway".TM.StepNo;
_00e: NOP   0;
      A     L 3.0;
      A     "DB_Steps"._BOOL.EMPTY_active;
      JNB   _00f;
      L     "DB_Steps"._INT.EMPTY_Steps;
      T     "DB_ComGateway".TM.StepNo;
_00f: NOP   0;
NETWORK
TITLE = Working Hours
      L     0;
      T     "DB_ComGateway".TM.WorkHours;
      NOP   0;
NETWORK
TITLE = Life counter
      A     "ON";
      =     L 3.0;
      A     L 3.0;
      JNB   _010;
      L     "DB_ComGateway".FM.CommCounterFromMaster;
      L     1;
      +I;
      T     "DB_ComGateway".TM.CommCounterToMaster;
_010: NOP   0;
      A     L 3.0;
      A(;
      L     "DB_ComGateway".FM.CommCounterFromMaster;
      L     9999;
      >I;
      );
      JNB   _011;
      L     1;
      T     "DB_ComGateway".TM.CommCounterToMaster;
_011: NOP   0;
      A     L 3.0;
      JNB   _012;
      L     "DB_ComGateway".TM.CommCounterToMaster;
      T     "DB_ComGateway".TM.Spare[5];
_012: NOP   0;
NETWORK
TITLE = BAUER
      A(;
      A(;
      L     W#16#4241;
      T     "DB_ComGateway".TM.Spare[1];
      SET;
      SAVE;
      CLR;
      A     BR;
      );
      JNB   _013;
      L     W#16#5545;
      T     "DB_ComGateway".TM.Spare[2];
      SET;
      SAVE;
      CLR;
_013: A     BR;
      );
      JNB   _014;
      L     W#16#5520;
      T     "DB_ComGateway".TM.Spare[3];
_014: NOP   0;
NETWORK
TITLE =
      A     "ON";
      SAVE;
END_FUNCTION

FUNCTION "STEPS_Control" : VOID	// FC 110
TITLE = Step Sequences
VERSION : 0.1
VAR_TEMP
  next : BOOL ;
  tmp_ActCircum : DINT ;
  tmp_CircumDiff : DINT ;
  tmp_OrderCircum : DINT ;
END_VAR
BEGIN
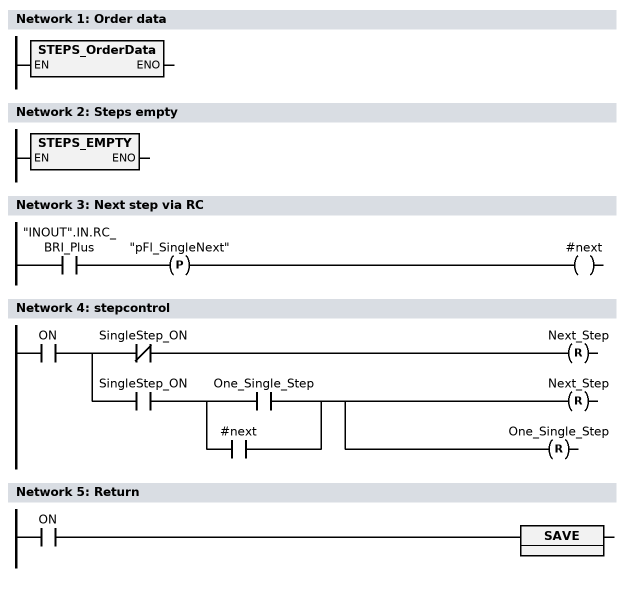
NETWORK
TITLE = Order data
      CALL  "STEPS_OrderData";
      NOP   0;
NETWORK
TITLE = Steps empty
      CALL  "STEPS_EMPTY";
      NOP   0;
NETWORK
TITLE = Next step via RC
      A     "INOUT".IN.RC_BRI_Plus;
      FP    "pFl_SingleNext";
      =     #next;
NETWORK
TITLE = stepcontrol
//Einzelschritt
      A     "ON";
      =     L 14.0;
      A     L 14.0;
      AN    "SingleStep_ON";
      R     "Next_Step";
      A     L 14.0;
      A     "SingleStep_ON";
      A(;
      O     "One_Single_Step";
      O     #next;
      );
      R     "Next_Step";
      R     "One_Single_Step";
NETWORK
TITLE = Return
      A     "ON";
      SAVE;
END_FUNCTION

FUNCTION "STEPS_OrderData" : VOID	// FC 111
TITLE = Steps OrderData
VERSION : 2.0
VAR_TEMP
  tmp_OrderPosValBRI : DINT ;
  tmp_di_1 : DINT ;
  tmp_di_DiffHoHu : DINT ;
  tmp_RetValErrCode : INT ;
  tmp_LifTargetPosNo : INT ;
  tmp_RetValErrCodeBRI : INT ;
  tmp_OrderPosNoBRI : INT ;
  tmp_OrderLIF_DBNo : INT ;
  tmp_OrderLIF_DBNo_2 : INT ;
  tmp_RetValErrBRI : BOOL ;
  tmp_BRI_DataOk : BOOL ;
  tmp_LIF_DataOK : BOOL ;
  tmp_TEL_DataOK : BOOL ;
  tmp_LifReleaseTarg : BOOL ;
  tmp_BriDataOK : BOOL ;
  tmp_LifTargetDataOK : BOOL ;
  tmp_OrderPosNoTRO : INT ;
  tmp_OrderPosValTRO : DINT ;
  tmp_TRBR : INT ;
  tmp_WID_DataOK : BOOL ;
  tmp_ReadDB_OK : BOOL ;
  tmp_StartDBCopy : BOOL ;
END_VAR
BEGIN
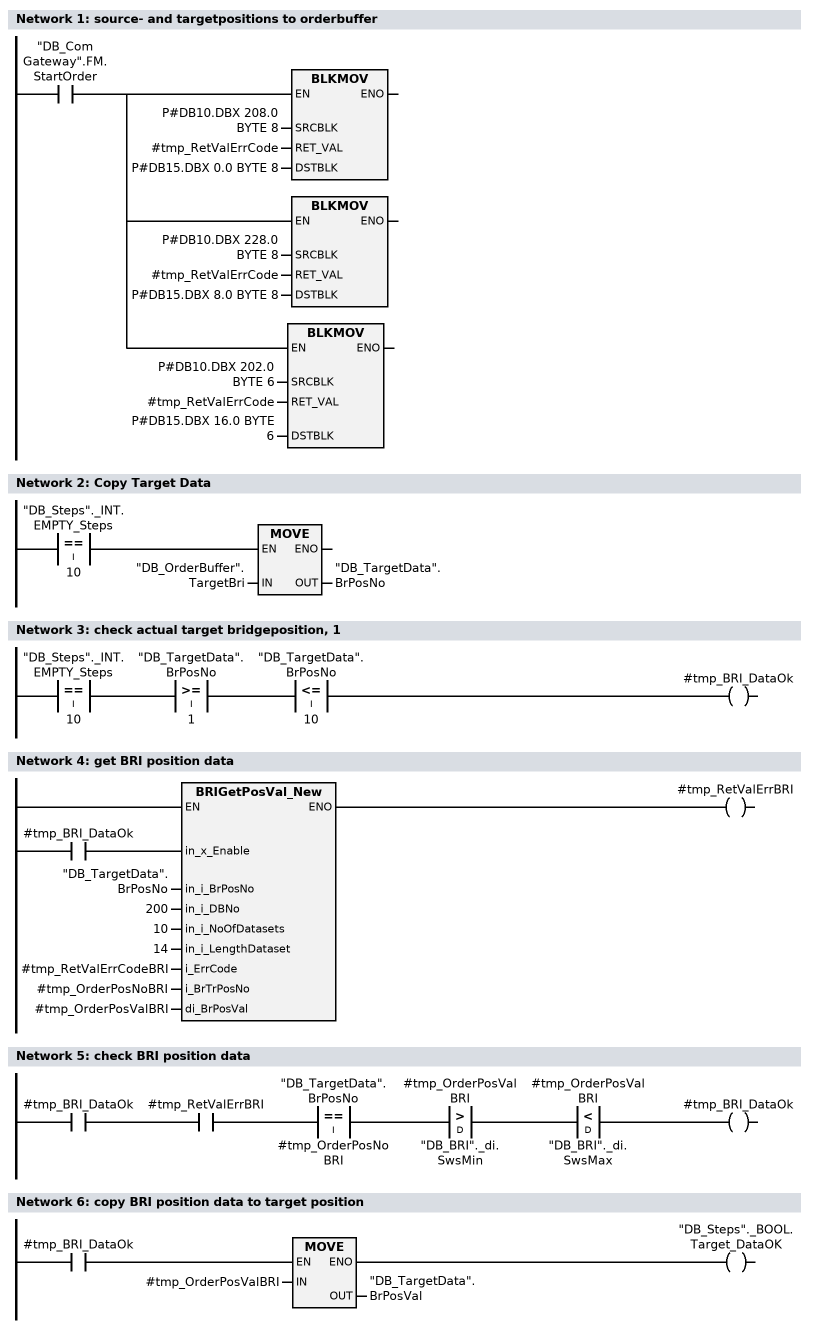
NETWORK
TITLE = source- and targetpositions to orderbuffer
      A     "DB_ComGateway".FM.StartOrder;
      =     L 35.0;
      A     L 35.0;
      JNB   _001;
      CALL  "BLKMOV" (
           SRCBLK                   := P#DB10.DBX 208.0 BYTE 8,
           RET_VAL                  := #tmp_RetValErrCode,
           DSTBLK                   := P#DB15.DBX 0.0 BYTE 8);
_001: NOP   0;
      A     L 35.0;
      JNB   _002;
      CALL  "BLKMOV" (
           SRCBLK                   := P#DB10.DBX 228.0 BYTE 8,
           RET_VAL                  := #tmp_RetValErrCode,
           DSTBLK                   := P#DB15.DBX 8.0 BYTE 8);
_002: NOP   0;
      A     L 35.0;
      JNB   _003;
      CALL  "BLKMOV" (
           SRCBLK                   := P#DB10.DBX 202.0 BYTE 6,
           RET_VAL                  := #tmp_RetValErrCode,
           DSTBLK                   := P#DB15.DBX 16.0 BYTE 6);
_003: NOP   0;
NETWORK
TITLE = Copy Target Data
      A(;
      L     "DB_Steps"._INT.EMPTY_Steps;
      L     10;
      ==I;
      );
      JNB   _004;
      L     "DB_OrderBuffer".TargetBri;
      T     "DB_TargetData".BrPosNo;
_004: NOP   0;
NETWORK
TITLE = check actual target bridgeposition, 1 
      A(;
      L     "DB_Steps"._INT.EMPTY_Steps;
      L     10;
      ==I;
      );
      A(;
      L     "DB_TargetData".BrPosNo;
      L     1;
      >=I;
      );
      A(;
      L     "DB_TargetData".BrPosNo;
      L     10;
      <=I;
      );
      =     #tmp_BRI_DataOk;
NETWORK
TITLE = get BRI position data
      A     #tmp_BRI_DataOk;
      =     L 35.0;
      BLD   103;
      CALL  "BRIGetPosVal_New" (
           in_x_Enable              := L 35.0,
           in_i_BrPosNo             := "DB_TargetData".BrPosNo,
           in_i_DBNo                := 200,
           in_i_NoOfDatasets        := 10,
           in_i_LengthDataset       := 14,
           i_ErrCode                := #tmp_RetValErrCodeBRI,
           i_BrTrPosNo              := #tmp_OrderPosNoBRI,
           di_BrPosVal              := #tmp_OrderPosValBRI);
      A     BR;
      =     #tmp_RetValErrBRI;
NETWORK
TITLE = check BRI position data
      A     #tmp_BRI_DataOk;
      A     #tmp_RetValErrBRI;
      A(;
      L     "DB_TargetData".BrPosNo;
      L     #tmp_OrderPosNoBRI;
      ==I;
      );
      A(;
      L     #tmp_OrderPosValBRI;
      L     "DB_BRI"._di.SwsMin;
      >D;
      );
      A(;
      L     #tmp_OrderPosValBRI;
      L     "DB_BRI"._di.SwsMax;
      <D;
      );
      =     #tmp_BRI_DataOk;
NETWORK
TITLE = copy BRI position data to target position
      A     #tmp_BRI_DataOk;
      JNB   _005;
      L     #tmp_OrderPosValBRI;
      T     "DB_TargetData".BrPosVal;
      SET;
      SAVE;
      CLR;
_005: A     BR;
      =     "DB_Steps"._BOOL.Target_DataOK;
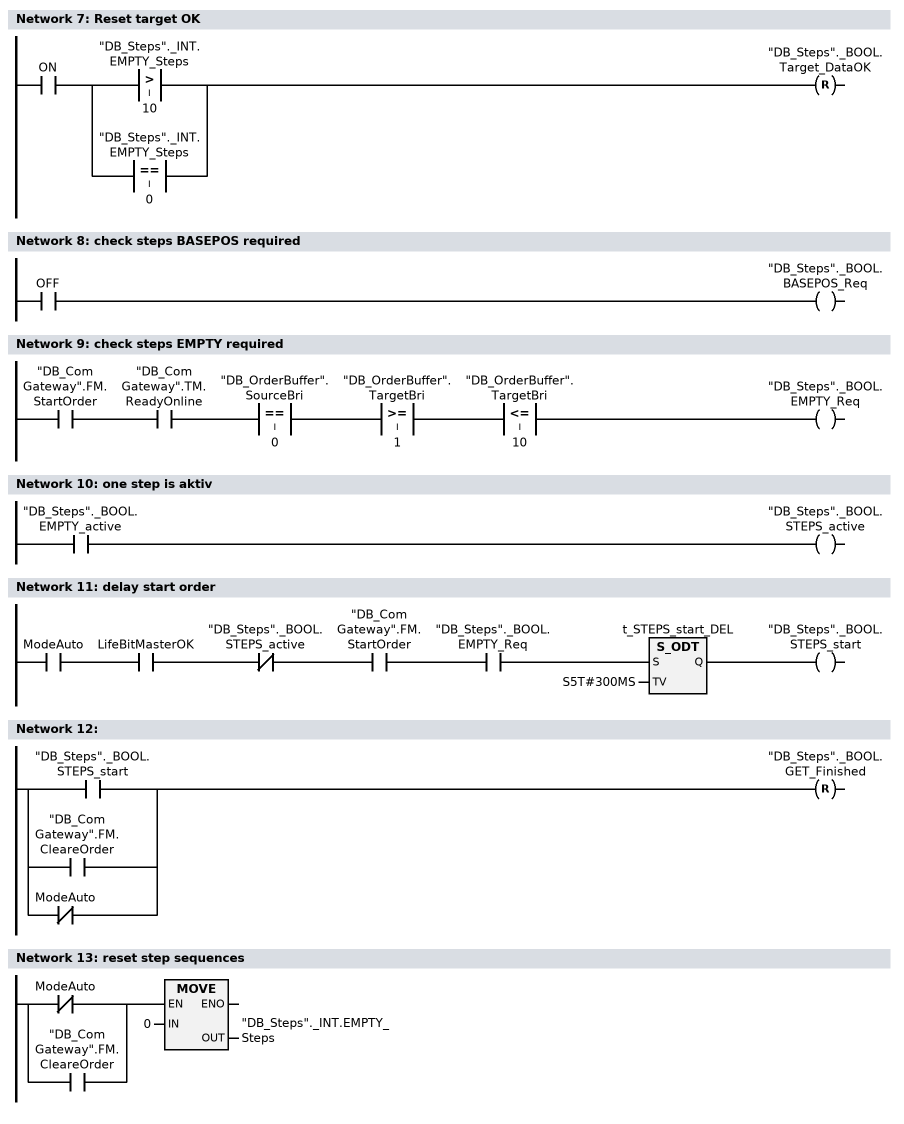
NETWORK
TITLE = Reset target OK
      A     "ON";
      A(;
      O(;
      L     "DB_Steps"._INT.EMPTY_Steps;
      L     10;
      >I;
      );
      O(;
      L     "DB_Steps"._INT.EMPTY_Steps;
      L     0;
      ==I;
      );
      );
      R     "DB_Steps"._BOOL.Target_DataOK;
NETWORK
TITLE = check steps BASEPOS required
      A     "OFF";
      =     "DB_Steps"._BOOL.BASEPOS_Req;
NETWORK
TITLE = check steps EMPTY required
      A     "DB_ComGateway".FM.StartOrder;
      A     "DB_ComGateway".TM.ReadyOnline;
      A(;
      L     "DB_OrderBuffer".SourceBri;
      L     0;
      ==I;
      );
      A(;
      L     "DB_OrderBuffer".TargetBri;
      L     1;
      >=I;
      );
      A(;
      L     "DB_OrderBuffer".TargetBri;
      L     10;
      <=I;
      );
      =     "DB_Steps"._BOOL.EMPTY_Req;
NETWORK
TITLE = one step is aktiv
      A     "DB_Steps"._BOOL.EMPTY_active;
      =     "DB_Steps"._BOOL.STEPS_active;
NETWORK
TITLE = delay start order
      A     "ModeAuto";
      A     "LifeBitMasterOK";
      AN    "DB_Steps"._BOOL.STEPS_active;
      A     "DB_ComGateway".FM.StartOrder;
      A     "DB_Steps"._BOOL.EMPTY_Req;
      L     S5T#300MS;
      SD    "t_STEPS_start_DEL";
      NOP   0;
      NOP   0;
      NOP   0;
      A     "t_STEPS_start_DEL";
      =     "DB_Steps"._BOOL.STEPS_start;
NETWORK
TITLE =
      O     "DB_Steps"._BOOL.STEPS_start;
      O     "DB_ComGateway".FM.CleareOrder;
      ON    "ModeAuto";
      R     "DB_Steps"._BOOL.GET_Finished;
NETWORK
TITLE = reset step sequences
      A(;
      ON    "ModeAuto";
      O     "DB_ComGateway".FM.CleareOrder;
      );
      JNB   _006;
      L     0;
      T     "DB_Steps"._INT.EMPTY_Steps;
_006: NOP   0;
